KUKA KRL data list: Rack_Verde_Abrir_PLC.dat

&ACCESS RVO1
&REL 186
&COMMENT ABRIR BAND RACK VERDE
&PARAM EDITMASK = *
&PARAM TEMPLATE = C:\KRC\Roboter\Template\vorgabe
&PARAM DISKPATH = KRC:\R1\Program\MAFELEC
DEFDAT  Rack_Verde_Abrir_PLC
;FOLD EXTERNAL DECLARATIONS;%{PE}%MKUKATPBASIS,%CEXT,%VCOMMON,%P
;FOLD GRIPPERTECH EXT
EXT  H50 (INT  :IN,INT  :IN,INT  :IN,GRP_TYP  :IN )
;ENDFOLD (GRIPPERTECH EXT)
;FOLD SPOTTECH EXT
EXT  USERSPOT (S_COMMAND  :IN,SPOT_TYPE  :IN )
;ENDFOLD (SPOTTECH EXT)
;FOLD BASISTECH EXT;%{PE}%MKUKATPBASIS,%CEXT,%VEXT,%P
EXT  BAS (BAS_COMMAND  :IN,REAL  :IN )
DECL INT SUCCESS
;ENDFOLD (BASISTECH EXT)
;FOLD USER EXT;%{E}%MKUKATPUSER,%CEXT,%VEXT,%P
;Make your modifications here

;ENDFOLD (USER EXT)
;ENDFOLD (EXTERNAL DECLARATIONS)
DECL BASIS_SUGG_T LAST_BASIS={POINT1[] "P0                      ",POINT2[] "P0                      ",CP_PARAMS[] "CPDAT0                  ",PTP_PARAMS[] "PDAT0                   ",CONT[] "                        ",CP_VEL[] "2                       ",PTP_VEL[] " 100                    ",SYNC_PARAMS[] "SYNCDAT                 ",SPL_NAME[] "S0                      ",A_PARAMS[] "ADAT0                   "}
DECL PDAT PH={VEL 100.000,ACC 100.000,APO_DIST 100.000,APO_MODE #CDIS,GEAR_JERK 50.0000,EXAX_IGN 0}
DECL E6POS XPOS_ESPERA_AREA1={X 112.943756,Y -227.851166,Z 2716.11304,A 36.2463837,B -15.5853510,C 56.0520973,S 3,T 42,E1 0.0,E2 0.0,E3 0.0,E4 0.0,E5 0.0,E6 0.0}
DECL FDAT FPOS_ESPERA_AREA1={TOOL_NO 9,BASE_NO 0,IPO_FRAME #BASE,POINT2[] " ",TQ_STATE FALSE}
DECL E6POS XAUX_ABRIR_B1={X 587.201599,Y -489.010620,Z -475.813660,A -88.3275681,B 24.5205555,C 90.7009506,S 6,T 58,E1 0.0,E2 0.0,E3 0.0,E4 0.0,E5 0.0,E6 0.0}
DECL E6POS XFIN_ABRIR_B1={X 586.228516,Y -669.031433,Z -259.029266,A -88.3565216,B 14.8194904,C 90.8183289,S 6,T 58,E1 0.0,E2 0.0,E3 0.0,E4 0.0,E5 0.0,E6 0.0}
DECL FDAT FFin_abrir_B1={TOOL_NO 2,BASE_NO 1,IPO_FRAME #BASE,POINT2[] "XAux_abrir_B1",TQ_STATE FALSE}
DECL LDAT LL={VEL 2.00000,ACC 25.0000,APO_DIST 25.0000,APO_FAC 50.0000,AXIS_VEL 100.000,AXIS_ACC 100.000,ORI_TYP #VAR,CIRC_TYP #BASE,JERK_FAC 50.0000,GEAR_JERK 50.0000,EXAX_IGN 0}
DECL E6POS XIni_Abrir_B1={X 593.427795,Y -368.612946,Z -1005.56824,A -87.3675156,B 34.2713966,C 92.0303879,S 6,T 58,E1 0.0,E2 0.0,E3 0.0,E4 0.0,E5 0.0,E6 0.0}
DECL FDAT FIni_Abrir_B1={TOOL_NO 2,BASE_NO 1,IPO_FRAME #BASE,POINT2[] " ",TQ_STATE FALSE}
DECL E6POS XIni_Abrir_B2={X 608.223267,Y -399.385956,Z -788.021118,A -87.5396500,B 30.5008068,C 91.8593445,S 6,T 58,E1 0.0,E2 0.0,E3 0.0,E4 0.0,E5 0.0,E6 0.0}
DECL FDAT FIni_Abrir_B2={TOOL_NO 2,BASE_NO 1,IPO_FRAME #BASE,POINT2[] " ",TQ_STATE FALSE}
DECL E6POS XIni_Abrir_B3={X 605.183289,Y -398.008423,Z -586.524719,A -88.7595062,B 30.4067383,C 90.2486267,S 6,T 58,E1 0.0,E2 0.0,E3 0.0,E4 0.0,E5 0.0,E6 0.0}
DECL FDAT FIni_Abrir_B3={TOOL_NO 2,BASE_NO 1,IPO_FRAME #BASE,POINT2[] " ",TQ_STATE FALSE}
DECL E6POS XIni_Abrir_B4={X 624.520874,Y -372.304596,Z -384.585,A -91.7077484,B 27.0395851,C 88.8544846,S 6,T 58,E1 0.0,E2 0.0,E3 0.0,E4 0.0,E5 0.0,E6 0.0}
DECL FDAT FIni_Abrir_B4={TOOL_NO 2,BASE_NO 1,IPO_FRAME #BASE,POINT2[] " ",TQ_STATE FALSE}
DECL E6POS XIni_Abrir_B5={X 901.585388,Y -191.617203,Z -190.010590,A -91.1728210,B 0.874125481,C 90.2115555,S 6,T 58,E1 0.0,E2 0.0,E3 0.0,E4 0.0,E5 0.0,E6 0.0}
DECL FDAT FIni_Abrir_B5={TOOL_NO 2,BASE_NO 1,IPO_FRAME #BASE,POINT2[] " ",TQ_STATE FALSE}
DECL E6POS XAux_abrir_B2={X 608.067688,Y -448.978790,Z -425.069458,A -87.9471588,B 28.1070080,C 91.1555939,S 6,T 58,E1 0.0,E2 0.0,E3 0.0,E4 0.0,E5 0.0,E6 0.0}
DECL E6POS XFin_abrir_B2={X 613.295044,Y -693.075134,Z -26.0282650,A -88.5897827,B 16.9574356,C 89.9685059,S 6,T 58,E1 0.0,E2 0.0,E3 0.0,E4 0.0,E5 0.0,E6 0.0}
DECL FDAT FFin_abrir_B2={TOOL_NO 2,BASE_NO 1,IPO_FRAME #BASE,POINT2[] "XAux_abrir_B2",TQ_STATE FALSE}
DECL E6POS XAux_abrir_B3={X 615.091675,Y -486.873108,Z -138.074326,A -88.6231461,B 20.4924870,C 90.6878204,S 6,T 58,E1 0.0,E2 0.0,E3 0.0,E4 0.0,E5 0.0,E6 0.0}
DECL E6POS XFin_abrir_B3={X 609.512512,Y -724.535400,Z 168.119400,A -88.5443497,B 11.4755363,C 90.9477081,S 6,T 58,E1 0.0,E2 0.0,E3 0.0,E4 0.0,E5 0.0,E6 0.0}
DECL FDAT FFin_abrir_B3={TOOL_NO 2,BASE_NO 1,IPO_FRAME #BASE,POINT2[] "XAux_abrir_B3",TQ_STATE FALSE}
DECL E6POS XAux_abrir_B4={X 632.938721,Y -528.271057,Z 147.159790,A -90.4987335,B 19.9364357,C 89.1931381,S 6,T 58,E1 0.0,E2 0.0,E3 0.0,E4 0.0,E5 0.0,E6 0.0}
DECL E6POS XFin_abrir_B4={X 639.312,Y -703.977478,Z 360.755463,A -89.9486,B 16.4602070,C 89.2945404,S 6,T 58,E1 0.0,E2 0.0,E3 0.0,E4 0.0,E5 0.0,E6 0.0}
DECL FDAT FFin_abrir_B4={TOOL_NO 2,BASE_NO 1,IPO_FRAME #BASE,POINT2[] "XAux_abrir_B4",TQ_STATE FALSE}
DECL E6POS XAux_abrir_B5={X 900.010681,Y -193.963440,Z 139.901840,A -90.4641495,B 28.6735859,C 89.9829559,S 6,T 26,E1 0.0,E2 0.0,E3 0.0,E4 0.0,E5 0.0,E6 0.0}
DECL E6POS XFin_abrir_B5={X 900.862488,Y -640.628052,Z 831.914856,A -89.0514755,B 32.2201576,C 89.4377899,S 6,T 26,E1 0.0,E2 0.0,E3 0.0,E4 0.0,E5 0.0,E6 0.0}
DECL FDAT FFin_abrir_B5={TOOL_NO 2,BASE_NO 1,IPO_FRAME #BASE,POINT2[] " ",TQ_STATE FALSE}
DECL E6POS XPOS_AREA1_LIBRE={X -250.533554,Y -43.6507149,Z 2716.11304,A -84.6604385,B 6.50295877,C 57.2217522,S 3,T 42,E1 0.0,E2 0.0,E3 0.0,E4 0.0,E5 0.0,E6 0.0}
DECL FDAT FPOS_AREA1_LIBRE={TOOL_NO 9,BASE_NO 0,IPO_FRAME #BASE,POINT2[] " ",TQ_STATE FALSE}
DECL E6POS XP111={X -1268.25977,Y -1488.91943,Z 479.113403,A -88.3003082,B 32.4766350,C 90.6096954,S 6,T 58,E1 0.0,E2 0.0,E3 0.0,E4 0.0,E5 0.0,E6 0.0}
DECL FDAT FP111={TOOL_NO 2,BASE_NO 0,IPO_FRAME #BASE,POINT2[] " ",TQ_STATE FALSE}
DECL E6POS XP510={X 699.073425,Y 157.382584,Z -207.307632,A -91.0988541,B 27.0961266,C 90.2740173,S 6,T 58,E1 0.0,E2 0.0,E3 0.0,E4 0.0,E5 0.0,E6 0.0}
DECL FDAT FP510={TOOL_NO 2,BASE_NO 1,IPO_FRAME #BASE,POINT2[] " ",TQ_STATE FALSE}
DECL E6POS XP520={X 598.759583,Y 37.4629440,Z -430.013275,A -91.6994858,B 27.0489426,C 88.8922501,S 6,T 58,E1 0.0,E2 0.0,E3 0.0,E4 0.0,E5 0.0,E6 0.0}
DECL FDAT FP520={TOOL_NO 2,BASE_NO 1,IPO_FRAME #BASE,POINT2[] " ",TQ_STATE FALSE}
DECL E6POS XP10={X 699.073425,Y 157.382584,Z -207.307632,A -91.0988541,B 27.0961266,C 90.2740173,S 6,T 58,E1 0.0,E2 0.0,E3 0.0,E4 0.0,E5 0.0,E6 0.0}
DECL FDAT FP10={TOOL_NO 2,BASE_NO 1,IPO_FRAME #BASE,POINT2[] " ",TQ_STATE FALSE}
DECL E6POS XP410={X 598.759583,Y 37.4629440,Z -430.013275,A -91.6994858,B 27.0489426,C 88.8922501,S 6,T 58,E1 0.0,E2 0.0,E3 0.0,E4 0.0,E5 0.0,E6 0.0}
DECL FDAT FP410={TOOL_NO 2,BASE_NO 1,IPO_FRAME #BASE,POINT2[] " ",TQ_STATE FALSE}
DECL E6POS XP310={X 605.449768,Y 11.9160767,Z -619.185730,A -88.7927856,B 27.1827526,C 90.1777420,S 6,T 58,E1 0.0,E2 0.0,E3 0.0,E4 0.0,E5 0.0,E6 0.0}
DECL FDAT FP310={TOOL_NO 2,BASE_NO 1,IPO_FRAME #BASE,POINT2[] " ",TQ_STATE FALSE}
DECL E6POS XP210={X 605.619263,Y -13.2147684,Z -875.790039,A -88.7865601,B 27.8310604,C 90.1928787,S 6,T 58,E1 0.0,E2 0.0,E3 0.0,E4 0.0,E5 0.0,E6 0.0}
DECL FDAT FP210={TOOL_NO 2,BASE_NO 1,IPO_FRAME #BASE,POINT2[] " ",TQ_STATE FALSE}
DECL E6POS XP110={X 608.377686,Y 9.23371887,Z -979.781311,A -88.1984787,B 29.7267971,C 91.1910172,S 6,T 58,E1 0.0,E2 0.0,E3 0.0,E4 0.0,E5 0.0,E6 0.0}
DECL FDAT FP110={TOOL_NO 2,BASE_NO 1,IPO_FRAME #BASE,POINT2[] " ",TQ_STATE FALSE}
DECL E6POS XP420={X 605.449768,Y 11.9160767,Z -619.185730,A -88.7927856,B 27.1827526,C 90.1777420,S 6,T 58,E1 0.0,E2 0.0,E3 0.0,E4 0.0,E5 0.0,E6 0.0}
DECL FDAT FP420={TOOL_NO 2,BASE_NO 1,IPO_FRAME #BASE,POINT2[] " ",TQ_STATE FALSE}
DECL E6POS XP320={X 605.619263,Y -13.2147684,Z -875.790039,A -88.7865601,B 27.8310604,C 90.1928787,S 6,T 58,E1 0.0,E2 0.0,E3 0.0,E4 0.0,E5 0.0,E6 0.0}
DECL FDAT FP320={TOOL_NO 2,BASE_NO 1,IPO_FRAME #BASE,POINT2[] " ",TQ_STATE FALSE}
DECL E6POS XP220={X 608.377686,Y 9.23371887,Z -979.781311,A -88.1984787,B 29.7267971,C 91.1910172,S 6,T 58,E1 0.0,E2 0.0,E3 0.0,E4 0.0,E5 0.0,E6 0.0}
DECL FDAT FP220={TOOL_NO 2,BASE_NO 1,IPO_FRAME #BASE,POINT2[] " ",TQ_STATE FALSE}
DECL E6POS XP120={X 699.073425,Y 157.382584,Z -207.307632,A -91.0988541,B 27.0961266,C 90.2740173,S 6,T 58,E1 0.0,E2 0.0,E3 0.0,E4 0.0,E5 0.0,E6 0.0}
DECL FDAT FP120={TOOL_NO 2,BASE_NO 1,IPO_FRAME #BASE,POINT2[] " ",TQ_STATE FALSE}
DECL E6POS XP121={X 444.231262,Y 453.996155,Z 946.107,A -102.024231,B -19.0647125,C 118.088737,S 2,T 42,E1 0.0,E2 0.0,E3 0.0,E4 0.0,E5 0.0,E6 0.0}
DECL FDAT FP121={TOOL_NO 2,BASE_NO 1,IPO_FRAME #BASE,POINT2[] " ",TQ_STATE FALSE}
DECL E6POS XP_ABRIR10={X 1867.18530,Y 204.510223,Z 1473.97632,A -84.6604385,B 6.50295877,C 57.2217522,S 3,T 42,E1 0.0,E2 0.0,E3 0.0,E4 0.0,E5 0.0,E6 0.0}
DECL FDAT FP_ABRIR10={TOOL_NO 2,BASE_NO 1,IPO_FRAME #BASE,POINT2[] " ",TQ_STATE FALSE}
DECL E6POS XP_AHOME={X 112.943756,Y -227.851166,Z 2716.11304,A 36.2463837,B -15.5853510,C 56.0520973,S 3,T 42,E1 0.0,E2 0.0,E3 0.0,E4 0.0,E5 0.0,E6 0.0}
DECL FDAT FP_aHOME={TOOL_NO 9,BASE_NO 0,IPO_FRAME #BASE,POINT2[] " ",TQ_STATE FALSE}
DECL E6POS XP11={X 500.256653,Y 161.434937,Z -226.642746,A -88.9033661,B 31.1327610,C 89.4967575,S 6,T 58,E1 0.0,E2 0.0,E3 0.0,E4 0.0,E5 0.0,E6 0.0}
DECL FDAT FP11={TOOL_NO 2,BASE_NO 1,IPO_FRAME #BASE,POINT2[] " ",TQ_STATE FALSE}
DECL E6POS XP0={X 549.337402,Y 294.945343,Z -525.939819,A -88.6139679,B 32.7546692,C 89.9199066,S 6,T 58,E1 0.0,E2 0.0,E3 0.0,E4 0.0,E5 0.0,E6 0.0}
DECL FDAT FP0={TOOL_NO 2,BASE_NO 1,IPO_FRAME #BASE,POINT2[] " ",TQ_STATE FALSE}
DECL LDAT LCPDAT1={VEL 2.00000,ACC 25.0000,APO_DIST 100.000,APO_FAC 50.0000,AXIS_VEL 100.000,AXIS_ACC 100.000,ORI_TYP #VAR,CIRC_TYP #BASE,JERK_FAC 50.0000,GEAR_JERK 50.0000,EXAX_IGN 0}
DECL PDAT PPDAT1={VEL 100.000,ACC 100.000,APO_DIST 100.000,GEAR_JERK 50.0000,EXAX_IGN 0}
DECL E6POS XP112211={X 548.096252,Y 56.0438080,Z -488.650848,A -88.5563202,B 27.2481651,C 89.8798828,S 6,T 58,E1 0.0,E2 0.0,E3 0.0,E4 0.0,E5 0.0,E6 0.0}
DECL FDAT FP112211={TOOL_NO 2,BASE_NO 1,IPO_FRAME #BASE,POINT2[] " ",TQ_STATE FALSE}
DECL PDAT PPDAT2={VEL 100.000,ACC 100.000,APO_DIST 100.000,GEAR_JERK 50.0000,EXAX_IGN 0}
DECL PDAT PPDAT3={VEL 100.000,ACC 100.000,APO_DIST 100.000,GEAR_JERK 50.0000,EXAX_IGN 0}
DECL PDAT PPDAT4={VEL 100.000,ACC 100.000,APO_DIST 100.000,GEAR_JERK 50.0000,EXAX_IGN 0}
DECL E6POS XP_FIN_ABRIR_B1={X 515.739929,Y 203.106186,Z -802.900696,A -88.4565048,B 31.1992207,C 90.3611603,S 6,T 58,E1 0.0,E2 0.0,E3 0.0,E4 0.0,E5 0.0,E6 0.0}
DECL FDAT FP_FIN_ABRIR_B1={TOOL_NO 2,BASE_NO 1,IPO_FRAME #BASE,POINT2[] " ",TQ_STATE FALSE}
DECL LDAT LH={VEL 2.00000,ACC 100.000,APO_DIST 100.000,APO_FAC 50.0000,AXIS_VEL 100.000,AXIS_ACC 100.000,ORI_TYP #VAR,CIRC_TYP #BASE,JERK_FAC 50.0000,GEAR_JERK 50.0000,EXAX_IGN 0}
DECL E6POS XPOS_ESCAPE={X 628.910095,Y 161.465546,Z -226.931656,A -88.8999939,B 31.1314793,C 89.4971771,S 6,T 58,E1 0.0,E2 0.0,E3 0.0,E4 0.0,E5 0.0,E6 0.0}
DECL FDAT FPOS_ESCAPE={TOOL_NO 2,BASE_NO 1,IPO_FRAME #BASE,POINT2[] " ",TQ_STATE FALSE}
DECL PDAT PPDAT5={VEL 100.000,ACC 100.000,APO_DIST 100.000,GEAR_JERK 50.0000,EXAX_IGN 0}
DECL LDAT LM={VEL 2.00000,ACC 35.0000,APO_DIST 25.0000,APO_FAC 50.0000,AXIS_VEL 100.000,AXIS_ACC 100.000,ORI_TYP #VAR,CIRC_TYP #BASE,JERK_FAC 50.0000,GEAR_JERK 50.0000,EXAX_IGN 0}
DECL FDAT FAux_abrir_B5={TOOL_NO 2,BASE_NO 1,IPO_FRAME #BASE,POINT2[] " ",TQ_STATE FALSE}
DECL LDAT LCPDAT2={VEL 2.00000,ACC 35.0000,APO_DIST 25.0000,APO_FAC 50.0000,AXIS_VEL 100.000,AXIS_ACC 100.000,ORI_TYP #VAR,CIRC_TYP #BASE,JERK_FAC 50.0000,GEAR_JERK 50.0000,EXAX_IGN 0}
DECL E6POS XAUX_ABRIR_B6={X 901.292236,Y -192.831421,Z -109.460472,A -91.1771,B -0.570868790,C 90.2113953,S 6,T 58,E1 0.0,E2 0.0,E3 0.0,E4 0.0,E5 0.0,E6 0.0}
DECL FDAT FAux_abrir_B6={TOOL_NO 2,BASE_NO 1,IPO_FRAME #BASE,POINT2[] " ",TQ_STATE FALSE}
DECL E6POS XAUX_ABRIR_B7={X 900.230,Y -244.949677,Z 260.172089,A -90.2476730,B 29.2348175,C 89.8884811,S 6,T 26,E1 0.0,E2 0.0,E3 0.0,E4 0.0,E5 0.0,E6 0.0}
DECL FDAT FAux_abrir_B7={TOOL_NO 2,BASE_NO 1,IPO_FRAME #BASE,POINT2[] " ",TQ_STATE FALSE}
DECL E6POS XAUX_ABRIR_B8={X 900.378296,Y -332.695374,Z 424.729156,A -89.9331589,B 30.0387497,C 89.7583694,S 6,T 26,E1 0.0,E2 0.0,E3 0.0,E4 0.0,E5 0.0,E6 0.0}
DECL FDAT FAux_abrir_B8={TOOL_NO 2,BASE_NO 1,IPO_FRAME #BASE,POINT2[] " ",TQ_STATE FALSE}
DECL E6POS XAUX_ABRIR_B9={X 865.439514,Y -125.572861,Z -227.929825,A -91.1604691,B 5.58096313,C 90.2201614,S 6,T 58,E1 0.0,E2 0.0,E3 0.0,E4 0.0,E5 0.0,E6 0.0}
DECL FDAT FAux_abrir_B9={TOOL_NO 2,BASE_NO 1,IPO_FRAME #BASE,POINT2[] " ",TQ_STATE FALSE}
DECL E6POS XP1={X 699.073425,Y 157.382584,Z -207.307632,A -91.0988541,B 27.0961266,C 90.2740173,S 6,T 58,E1 0.0,E2 0.0,E3 0.0,E4 0.0,E5 0.0,E6 0.0}
DECL FDAT FP1={TOOL_NO 2,BASE_NO 1,IPO_FRAME #BASE,POINT2[] " ",TQ_STATE FALSE}
DECL E6POS XAux_abrir_B10={X 1217.66492,Y -125.227119,Z -228.184372,A -76.0477,B 5.56443787,C 90.2668304,S 6,T 58,E1 0.0,E2 0.0,E3 0.0,E4 0.0,E5 0.0,E6 0.0}
DECL FDAT FAux_abrir_B10={TOOL_NO 2,BASE_NO 1,IPO_FRAME #BASE,POINT2[] " ",TQ_STATE FALSE}
DECL E6POS XIni_Abrir_B6={X 1240.70728,Y -191.182587,Z -190.294601,A -74.9191666,B 0.903282344,C 90.1932,S 6,T 58,E1 0.0,E2 0.0,E3 0.0,E4 0.0,E5 0.0,E6 0.0}
DECL FDAT FIni_Abrir_B6={TOOL_NO 2,BASE_NO 1,IPO_FRAME #BASE,POINT2[] " ",TQ_STATE FALSE}
DECL E6POS XAux_abrir_B11={X 1241.51563,Y -192.831421,Z -109.460472,A -76.1411438,B -0.570868671,C 90.2113953,S 6,T 58,E1 0.0,E2 0.0,E3 0.0,E4 0.0,E5 0.0,E6 0.0}
DECL FDAT FAux_abrir_B11={TOOL_NO 2,BASE_NO 1,IPO_FRAME #BASE,POINT2[] " ",TQ_STATE FALSE}
DECL E6POS XAux_abrir_B12={X 1216.66040,Y -193.931335,Z 139.882233,A -77.1661224,B 28.6737461,C 89.9869,S 6,T 26,E1 0.0,E2 0.0,E3 0.0,E4 0.0,E5 0.0,E6 0.0}
DECL FDAT FAux_abrir_B12={TOOL_NO 2,BASE_NO 1,IPO_FRAME #BASE,POINT2[] " ",TQ_STATE FALSE}
DECL E6POS XAux_abrir_B13={X 1228.16455,Y -244.842178,Z 260.123505,A -75.2080383,B 29.2341309,C 89.8981323,S 6,T 26,E1 0.0,E2 0.0,E3 0.0,E4 0.0,E5 0.0,E6 0.0}
DECL FDAT FAux_abrir_B13={TOOL_NO 2,BASE_NO 1,IPO_FRAME #BASE,POINT2[] " ",TQ_STATE FALSE}
DECL E6POS XAux_abrir_B14={X 1244.98633,Y -332.694550,Z 424.729645,A -77.6737900,B 30.0387135,C 89.7583237,S 6,T 26,E1 0.0,E2 0.0,E3 0.0,E4 0.0,E5 0.0,E6 0.0}
DECL FDAT FAux_abrir_B14={TOOL_NO 2,BASE_NO 1,IPO_FRAME #BASE,POINT2[] " ",TQ_STATE FALSE}
DECL E6POS XFin_abrir_B6={X 1205.18689,Y -640.627258,Z 831.915955,A -72.7500687,B 32.2200928,C 89.4376831,S 6,T 26,E1 0.0,E2 0.0,E3 0.0,E4 0.0,E5 0.0,E6 0.0}
DECL FDAT FFin_abrir_B6={TOOL_NO 2,BASE_NO 1,IPO_FRAME #BASE,POINT2[] " ",TQ_STATE FALSE}
DECL E6POS XP1_new={X 699.073425,Y 157.382584,Z -207.307632,A -91.0988541,B 27.0961266,C 90.2740173,S 6,T 58,E1 0.0,E2 0.0,E3 0.0,E4 0.0,E5 0.0,E6 0.0}
DECL FDAT FP1_new={TOOL_NO 2,BASE_NO 1,IPO_FRAME #BASE,POINT2[] " ",TQ_STATE FALSE}
DECL E6POS XP2_NEW={X 1217.66492,Y -125.227119,Z -228.184372,A -76.0477,B 5.56443787,C 90.2668304,S 6,T 58,E1 0.0,E2 0.0,E3 0.0,E4 0.0,E5 0.0,E6 0.0}
DECL FDAT Fp2_new={TOOL_NO 2,BASE_NO 1,IPO_FRAME #BASE,POINT2[] " ",TQ_STATE FALSE}
DECL E6POS XP2={X 1217.66492,Y -125.227119,Z -228.184372,A -76.0477,B 5.56443787,C 90.2668304,S 6,T 58,E1 0.0,E2 0.0,E3 0.0,E4 0.0,E5 0.0,E6 0.0}
DECL FDAT FP2={TOOL_NO 2,BASE_NO 1,IPO_FRAME #BASE,POINT2[] " ",TQ_STATE FALSE}
DECL LDAT LCPDAT3={VEL 2.00000,ACC 35.0000,APO_DIST 25.0000,APO_FAC 50.0000,AXIS_VEL 100.000,AXIS_ACC 100.000,ORI_TYP #VAR,CIRC_TYP #BASE,JERK_FAC 50.0000,GEAR_JERK 50.0000,EXAX_IGN 0}
DECL E6POS XP3={X 699.073425,Y 157.382584,Z -207.307632,A -91.0988541,B 27.0961266,C 90.2740173,S 6,T 58,E1 0.0,E2 0.0,E3 0.0,E4 0.0,E5 0.0,E6 0.0}
DECL FDAT FP3={TOOL_NO 2,BASE_NO 1,IPO_FRAME #BASE,POINT2[] " ",TQ_STATE FALSE}
DECL LDAT LCPDAT4={VEL 2.00000,ACC 35.0000,APO_DIST 100.000,APO_FAC 50.0000,AXIS_VEL 100.000,AXIS_ACC 100.000,ORI_TYP #VAR,CIRC_TYP #BASE,JERK_FAC 50.0000,GEAR_JERK 50.0000,EXAX_IGN 0}
DECL E6POS XP4={X 1240.70728,Y -191.182587,Z -190.294601,A -74.9191666,B 0.903282344,C 90.1932,S 6,T 58,E1 0.0,E2 0.0,E3 0.0,E4 0.0,E5 0.0,E6 0.0}
DECL FDAT FP4={TOOL_NO 2,BASE_NO 1,IPO_FRAME #BASE,POINT2[] " ",TQ_STATE FALSE}
DECL LDAT LCPDAT5={VEL 2.00000,ACC 35.0000,APO_DIST 25.0000,APO_FAC 50.0000,AXIS_VEL 100.000,AXIS_ACC 100.000,ORI_TYP #VAR,CIRC_TYP #BASE,JERK_FAC 50.0000,GEAR_JERK 50.0000,EXAX_IGN 0}
DECL E6POS XP5={X 1241.51563,Y -192.831421,Z -109.460472,A -76.1411438,B -0.570868671,C 90.2113953,S 6,T 58,E1 0.0,E2 0.0,E3 0.0,E4 0.0,E5 0.0,E6 0.0}
DECL FDAT FP5={TOOL_NO 2,BASE_NO 1,IPO_FRAME #BASE,POINT2[] " ",TQ_STATE FALSE}
DECL LDAT LCPDAT6={VEL 2.00000,ACC 35.0000,APO_DIST 25.0000,APO_FAC 50.0000,AXIS_VEL 100.000,AXIS_ACC 100.000,ORI_TYP #VAR,CIRC_TYP #BASE,JERK_FAC 50.0000,GEAR_JERK 50.0000,EXAX_IGN 0}
DECL E6POS XP6={X 1216.66040,Y -193.931335,Z 139.882233,A -77.1661224,B 28.6737461,C 89.9869,S 6,T 26,E1 0.0,E2 0.0,E3 0.0,E4 0.0,E5 0.0,E6 0.0}
DECL FDAT FP6={TOOL_NO 2,BASE_NO 1,IPO_FRAME #BASE,POINT2[] " ",TQ_STATE FALSE}
DECL LDAT LCPDAT7={VEL 2.00000,ACC 35.0000,APO_DIST 25.0000,APO_FAC 50.0000,AXIS_VEL 100.000,AXIS_ACC 100.000,ORI_TYP #VAR,CIRC_TYP #BASE,JERK_FAC 50.0000,GEAR_JERK 50.0000,EXAX_IGN 0}
DECL E6POS XP7={X 1228.16455,Y -244.842178,Z 260.123505,A -75.2080383,B 29.2341309,C 89.8981323,S 6,T 26,E1 0.0,E2 0.0,E3 0.0,E4 0.0,E5 0.0,E6 0.0}
DECL FDAT FP7={TOOL_NO 2,BASE_NO 1,IPO_FRAME #BASE,POINT2[] " ",TQ_STATE FALSE}
DECL LDAT LCPDAT8={VEL 2.00000,ACC 35.0000,APO_DIST 25.0000,APO_FAC 50.0000,AXIS_VEL 100.000,AXIS_ACC 100.000,ORI_TYP #VAR,CIRC_TYP #BASE,JERK_FAC 50.0000,GEAR_JERK 50.0000,EXAX_IGN 0}
DECL E6POS XP8={X 1244.98633,Y -332.694550,Z 424.729645,A -77.6737900,B 30.0387135,C 89.7583237,S 6,T 26,E1 0.0,E2 0.0,E3 0.0,E4 0.0,E5 0.0,E6 0.0}
DECL FDAT FP8={TOOL_NO 2,BASE_NO 1,IPO_FRAME #BASE,POINT2[] " ",TQ_STATE FALSE}
DECL LDAT LCPDAT9={VEL 2.00000,ACC 35.0000,APO_DIST 25.0000,APO_FAC 50.0000,AXIS_VEL 100.000,AXIS_ACC 100.000,ORI_TYP #VAR,CIRC_TYP #BASE,JERK_FAC 50.0000,GEAR_JERK 50.0000,EXAX_IGN 0}
DECL E6POS XP9={X 1205.18689,Y -640.627258,Z 831.915955,A -72.7500687,B 32.2200928,C 89.4376831,S 6,T 26,E1 0.0,E2 0.0,E3 0.0,E4 0.0,E5 0.0,E6 0.0}
DECL FDAT FP9={TOOL_NO 2,BASE_NO 1,IPO_FRAME #BASE,POINT2[] " ",TQ_STATE FALSE}
DECL LDAT LCPDAT10={VEL 2.00000,ACC 35.0000,APO_DIST 25.0000,APO_FAC 50.0000,AXIS_VEL 100.000,AXIS_ACC 100.000,ORI_TYP #VAR,CIRC_TYP #BASE,JERK_FAC 50.0000,GEAR_JERK 50.0000,EXAX_IGN 0}
ENDDAT
